FUNCTION_BLOCK FB_Door
VAR
	Actor AT %Q*:BOOL;
	Sensor AT %I*:BOOL;
END_VAR

METHOD Close : BOOL
VAR_INPUT
END_VAR
Actor:=false;
END_METHOD

METHOD isLocked : BOOL
VAR_INPUT
END_VAR
IF NOT actor AND sensor THEN
	isLocked:=TRUE;
ELSE
	isLocked:=FALSE;
END_IF
END_METHOD

METHOD Open : BOOL
VAR_INPUT
END_VAR
Actor:=true;
END_METHOD

METHOD Toggle : BOOL
VAR_INPUT
END_VAR
Actor:=not actor;
END_METHOD

END_FUNCTION_BLOCK

(* stored: Version 1.1.0.1, ProductVersion 3.1.4022.9
   POU FB_Door: Id {13b8ed84-3df6-4be1-a365-da4e090bc978}, SpecialFunc None
   Method Close: Id {9303b82d-af39-49d7-b61b-2b5583551cd0}
   Method isLocked: Id {268a71b7-8e62-40bb-ba2d-da39eaa4695e}
   Method Open: Id {e621c13a-faf3-45f9-91fa-1f05c55c12b4}
   Method Toggle: Id {f0309b50-75fd-4a13-bcc1-544d21e78956} *)
